% RSLogix 500 project RETTND.RSS, saved by version 9.00.00.04 %
PROJECT "UNTITLED"    % processor: Bul.1763 MicroLogix 1100 Series B %

PROGRAM FILES
  LAD 2   6 rungs
  LAD 3 "SUBROUTINE"  6 rungs

DATA FILES
  O0 OUTPUT  4 elements
  I1 INPUT  6 elements
  S2 STATUS  66 elements
  B3 BINARY  4 elements
  T4 TIMER  1 elements
  C5 COUNTER  1 elements
  R6 CONTROL  1 elements
  N7 INTEGER  3 elements
  F8 FLOAT  1 elements

LADDER 2
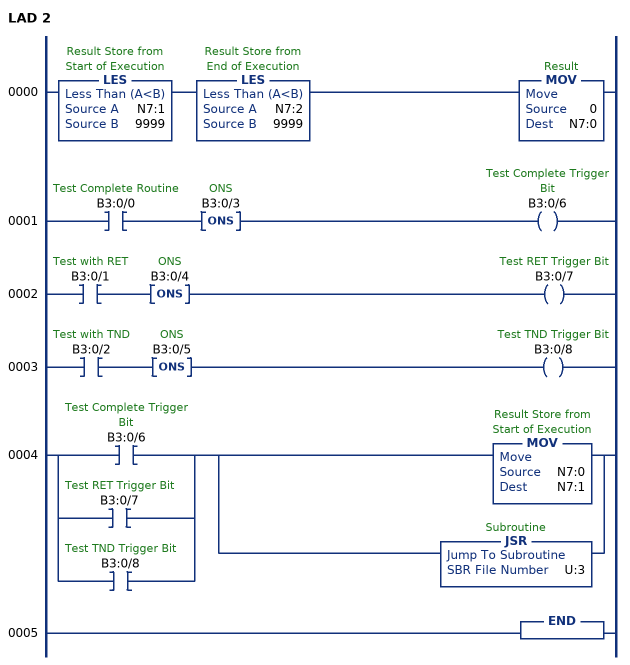
% Rung: 0 %
SOR LES N7:1 9999 LES N7:2 9999 MOV 0 N7:0 EOR
%   N7:1  "Result Store from Start of Execution" %
%   N7:2  "Result Store from End of Execution" %
%   N7:0  "Result" %
% Rung: 1 %
SOR XIC B3:0/0 ONS B3:0/3 OTE B3:0/6 EOR
%   B3:0/0  "Test Complete Routine" %
%   B3:0/3  "ONS" %
%   B3:0/6  "Test Complete Trigger Bit" %
% Rung: 2 %
SOR XIC B3:0/1 ONS B3:0/4 OTE B3:0/7 EOR
%   B3:0/1  "Test with RET" %
%   B3:0/4  "ONS" %
%   B3:0/7  "Test RET Trigger Bit" %
% Rung: 3 %
SOR XIC B3:0/2 ONS B3:0/5 OTE B3:0/8 EOR
%   B3:0/2  "Test with TND" %
%   B3:0/5  "ONS" %
%   B3:0/8  "Test TND Trigger Bit" %
% Rung: 4 %
SOR BST XIC B3:0/6 NXB XIC B3:0/7 NXB XIC B3:0/8 BND BST MOV N7:0 N7:1 NXB JSR U:3 BND EOR
%   B3:0/6  "Test Complete Trigger Bit" %
%   B3:0/7  "Test RET Trigger Bit" %
%   B3:0/8  "Test TND Trigger Bit" %
%   N7:0  "Result" %
%   N7:1  "Result Store from Start of Execution" %
%   U:3  "Subroutine" %
% Rung: 5 %
SOR END EOR

LADDER 3 "SUBROUTINE"
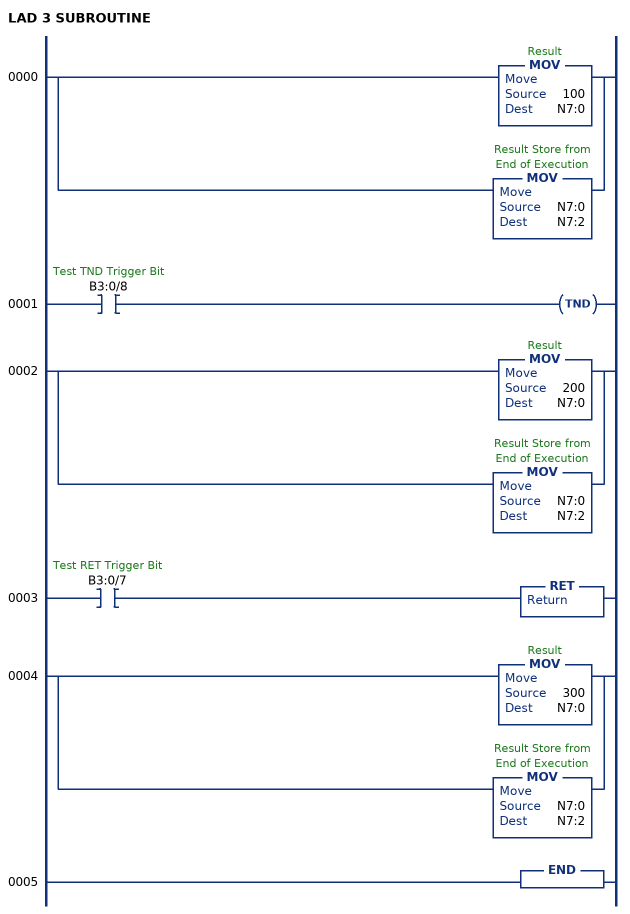
% Rung: 0 %
SOR BST MOV 100 N7:0 NXB MOV N7:0 N7:2 BND EOR
%   N7:0  "Result" %
%   N7:2  "Result Store from End of Execution" %
% Rung: 1 %
SOR XIC B3:0/8 TND EOR
%   B3:0/8  "Test TND Trigger Bit" %
% Rung: 2 %
SOR BST MOV 200 N7:0 NXB MOV N7:0 N7:2 BND EOR
%   N7:0  "Result" %
%   N7:2  "Result Store from End of Execution" %
% Rung: 3 %
SOR XIC B3:0/7 RET EOR
%   B3:0/7  "Test RET Trigger Bit" %
% Rung: 4 %
SOR BST MOV 300 N7:0 NXB MOV N7:0 N7:2 BND EOR
%   N7:0  "Result" %
%   N7:2  "Result Store from End of Execution" %
% Rung: 5 %
SOR END EOR

OTHER DOCUMENTED ADDRESSES
  B3:0  "Static Word 1"
  B3:1  "Static Word 2"
  B3:2  "Result Word"
  B3:3/0  "NOT Test button"
  B3:3/1  "AND Test button"
  B3:3/2  "OR Test button"
  B3:3/3  "CLR Test button"
